TYPE ST_RejectReasonOUT1 :
STRUCT
	Reason	:STRING;
END_STRUCT
END_TYPE

(* stored: Version 1.1.0.1, ProductVersion 3.1.4024.13
   DUT ST_RejectReasonOUT1: Id {dd3619f1-bad2-4efa-b8b7-a28440bbca49} *)
